FUNCTION_BLOCK FB_TsConnection_State
VAR_INPUT
	nState	: USINT;
END_VAR
VAR_OUTPUT
	sState	: STRING;
END_VAR
VAR
END_VAR

CASE nState OF
		100:	sState := 'Reset state';
		101:	sState := 'Session state';
		102:	sState := 'Connection state';
		103:	sState := 'Parameter state';
		104:	sState := 'Data state';
		105:	sState := 'Shutdown state';
ELSE
	sState := 'unknown';
END_CASE

END_FUNCTION_BLOCK

(* stored: Version 1.1.0.1, ProductVersion 3.1.4024.15
   POU FB_TsConnection_State: Id {b9ca1766-7f9d-4df2-88c3-15076e53ef23}, SpecialFunc None *)
